INTERFACE ISignalLightsController

PROPERTY GetColorsSignalLightMachineModes : ColorsSignalLightMachineModes
GET
END_GET
END_PROPERTY

PROPERTY GetColorsSignalLightMachineStatus : ColorsSignalLightMachineModes
GET
END_GET
END_PROPERTY

METHOD SetBlinkTime
VAR_INPUT
	blinkTime : TIME ;
END_VAR
END_METHOD

METHOD SetMachineMode : ColorsSignalLightMachineModes
VAR_INPUT
    currentMachineMode : eMachineModes := eMachineModes.Idle;
END_VAR
END_METHOD

METHOD SetMachineStatusOff : ColorsSignalLightsStatus
VAR_INPUT
    currentMachineStatus : eMachineStatus ;
END_VAR
END_METHOD

METHOD SetMachineStatusOn : ColorsSignalLightsStatus
VAR_INPUT
    currentMachineStatus : eMachineStatus ;
END_VAR
END_METHOD

END_INTERFACE

(* stored: Version 1.1.0.1, ProductVersion 3.1.4024.12
   Itf ISignalLightsController: Id {5cc853b6-a6b4-052f-2580-1168e385b567}
   Property GetColorsSignalLightMachineModes: Id {38e34ed0-21eb-03eb-0c2c-f07eb4f78088}
   Get Get: Id {8b9b8ee7-4b0c-0379-1ae1-4eee6175b99a}
   Property GetColorsSignalLightMachineStatus: Id {0a127001-5391-07a4-1104-fe4e47abccef}
   Get Get: Id {681124da-3b80-0284-0316-ff0fa244f1cc}
   Method SetBlinkTime: Id {71c84436-d35b-0c87-0414-decff83dd88f}
   Method SetMachineMode: Id {362b10ad-363d-0e31-2181-9b66b7933c66}
   Method SetMachineStatusOff: Id {99d8ed84-32f0-0337-2bb7-ce97eb828066}
   Method SetMachineStatusOn: Id {34fa206c-f612-09fc-27dc-9eafa1f7979e} *)
